TYPE ST_DeviceOut :
STRUCT
	bRun	: BOOL; // on, off
	fValue	: LREAL; // override, power, ...
END_STRUCT
END_TYPE

(* stored: Version 1.1.0.1, ProductVersion 3.1.4024.12
   DUT ST_DeviceOut: Id {92bfada3-b042-49b1-b174-c9d01d71593b} *)
